(* Logix 5000 project; controller IF2_DEMO Emulate 5570 rev 20.12; software revision 20.04; part 2 of 8 *)
(* tags used below, declared in another part *)
   AlarmFillerConvJam : BOOL;
   ChangeOver_In_Progress : BOOL;
   Current_Order : STRING;
   CurrentCustomerName : STRING;
   CurrentPartName : STRING;
   DispenserLine : LineData;
   Filler_Stopped : BOOL;
   Labeler_Stopped : BOOL;
   Line1 : FTVPDemoLine;
   Next_Order : STRING;
   Next_Product : DINT;
   OEE_Part_Scrap_Old : DINT;
   OEE_Scrap_Filler : DINT;
   OrderQty : DINT[4];
   Packaging_Stopped : BOOL;
   PartCountRollOver : DINT;
   Previous_Order : STRING;
   PreviousCustomerName : STRING;
   PreviousPartName : STRING;
   ProdCounts : Counts;
   Product_Change : DINT;
   ProductionStart : BOOL;
   Starve_Block_Filler_Start_Toggle : BOOL;
   Starve_Block_Labeler_Start_Toggle : BOOL;
   Starve_Block_Packaging_Start_Toggle : BOOL;
   Timer1000ms : TIMER;
   Timer250ms : TIMER;
   WallClock : DINT[7];
   WC : WC[10];
   WorkOrder : WorkOrder;

PROGRAM FillerD   (* main routine MainRoutine *)
VAR
   Alarm_Filler1_Blocked : ALARM_DIGITAL;
   Alarm_Filler1_Starved : ALARM_DIGITAL;
   Alarm_Filler1_Stopped : ALARM_DIGITAL;
   ATest : BOOL;
   Block_Delay : TIMER := (PRE := 15000);
   Blocked_Condition : BOOL;
   Blocked_L : BOOL;
   BottleNum : STRING := '3';
   Change_Nextorder_name : BOOL;
   Change_order_name : BOOL;
   Ctrl_Bit : BOOL;
   DownStream_Run : ALIAS FOR WC[2].EventTrigger[0].1;
   DownStream_Running : ALIAS FOR WC[2].EventTrigger[0].8;
   Events : Events := (DownTime.Breakdown := 1, DownTime.BreakdownCode := 4, Control.StandbyCode := 1, Control.Auto := 1);
   Events_Control_Auto : ALIAS FOR WC_L.EventTrigger[0].5;
   Events_Control_OpStop : ALIAS FOR WC_L.EventTrigger[0].3;
   Events_Control_Run : ALIAS FOR WC_L.EventTrigger[0].1;
   Events_Control_Running : ALIAS FOR WC_L.EventTrigger[0].8;
   Events_Control_Standby : ALIAS FOR WC_L.EventTrigger[0].0;
   Events_Control_StandbyCode : ALIAS FOR WC_L.EventValue_REAL[1];
   Events_DownTime_Breakdown : ALIAS FOR WC_L.EventTrigger[0].2;
   Events_DownTime_BreakdownCode : ALIAS FOR WC_L.EventValue_REAL[2];
   Events_DownTime_Testing : ALIAS FOR WC_L.EventTrigger[0].7;
   Events_DownTime_UnschedMaint : ALIAS FOR WC_L.EventTrigger[0].6;
   Events_Operate_Load : ALIAS FOR WC_L.EventTrigger[0].10;
   Events_Operate_OrderProc : ALIAS FOR WC_L.EventTrigger[0].11;
   Events_Operate_Setup : ALIAS FOR WC_L.EventTrigger[0].9;
   Expected_Full_Production_Rate : DINT := 119;
   Filler : FTVPDemoWorkCell := (LineName := 'Line1', RunState := 1, Temperature := 95, ScrapRate := 6, ProductionRate := 119, Pressure := 123, OrderName := 'GF-08-CZ-525', CustomerName := 'Soda Inc.', PartName := 'GF-11');
   Filler_Start : BOOL := 1;
   Filler_State : DINT;
   Filler_Status : DINT := 1;
   Filler_Stop : BOOL;
   FillOunces : INT := 32;
   Force_Periodic_Changeover : DINT;
   HMI : HMIVars := (ScrapRate := 1.0, SpeedControl := 400.0, PrevSpeed := 100.0, CurrentProductionRate := 120.0, PartCountRollOver := 3500, MfgTimeBase := 1, MaxEventDur := 21.0, MinEventDur := 9.0, EventsPerHr := 100, EventDur := 20.688032, RunDur := 14.955534, MinRunDur := 5.0);
   MfgOrders : MfgOrders := (CustomerName := 'Big-Mart', OrderName := 'A123', ProdRate := 60.0, PartName := 'Apple-D12', WorkcellName := 'Filler 1', PartNameSav := 'Apple-D12');
   MfgOrders_CustomerName : ALIAS FOR WC_L.FlexSTRING[4];
   MfgOrders_Order : STRING := 'GF-08-CZ-525';
   MfgOrders_OrderName : ALIAS FOR WC_L.FlexSTRING[3];
   MfgOrders_OrderName_Blueberry : STRING := 'BL-03-RM-';
   MfgOrders_OrderName_Grapefruit : STRING := 'GF-08-CZ-';
   MfgOrders_OrderName_Kiwi : STRING := 'KW-05-JM-';
   MfgOrders_OrderName_Mango : STRING := 'MG-01-RZ-';
   MfgOrders_OrderNumber_Blueberry : DINT := 662;
   MfgOrders_OrderNumber_Grapefruit : DINT := 525;
   MfgOrders_OrderNumber_Kiwi : DINT := 651;
   MfgOrders_OrderNumber_Mango : DINT := 969;
   MfgOrders_OrderNumber_String : STRING := '970';
   MfgOrders_PartName : ALIAS FOR WC_L.FlexSTRING[0];
   Motion : DINT := 82;
   Motion_Counter : DINT := 1;
   Motion_Speed : DINT := 100;
   MotionCount : TIMER := (PRE := 9000, ACC := 8273, EN := 1, TT := 1);
   NA_Test : BOOL;
   New_Product_Change : BOOL;
   OEE : OEE := (IdealCycleTime := 5.0);
   OEE_IdealCycleTime : ALIAS FOR WC_L.IdealCT;
   OEE_Parts_Good : ALIAS FOR WC_L.GoodParts;
   OEE_Parts_Scrap : ALIAS FOR WC_L.ScrapParts;
   OEE_Parts_Total : ALIAS FOR WC_L.TotalParts;
   onsbits : DINT;
   OperatorID : ALIAS FOR WC_L.FlexREAL[1];
   Pressure1 : ALIAS FOR WC_L.PV[0];   // PSI
   ProductColor : DINT := 1;
   ProductColor_Save : DINT := 1;
   ProductColorCode : INT;
   RecipeFlag : BOOL;
   RecipeName : STRING := 'Super';
   SIM : SimVars := (Run.PRE := 14956, Event.PRE := 9000, Setup.PRE := 9000, Good := 2589.8208, Scrap := 26.160408, EventNumber := 11, UtilityBool[1] := 1, UtilityBool[2] := 1);
        .UTILITYBOOL[0]   // Enter Auto Mode ONS
        .UTILITYBOOL[1]   // Work Order Complete ONS
        .UTILITYBOOL[2]   // First Scan Bit
   skip : BOOL;
   Starve_Block_Filler_ONS : BOOL;
   Starve_Delay : TIMER := (PRE := 15000);
   Starved_L : BOOL;
   StateValue : ALIAS FOR WC_L.MonitorValue[0];
   Suppress : Events;
   Temperature1 : ALIAS FOR WC_L.PV[1];   // DEG
   TempReadTrigger : TIMER := (PRE := 5000, ACC := 3633, EN := 1, TT := 1);
   TempTimer : TIMER := (PRE := 10000, ACC := 3708, EN := 1, TT := 1);
   TempTimer2 : TIMER := (PRE := 5000, ACC := 3633, EN := 1, TT := 1);
   UpStream_Run : BOOL := 1;
   UpStream_Running : BOOL := 1;   // Not used-no upstream wc
   WC_L : ALIAS FOR WC[0];
END_VAR

ROUTINE MainRoutine   (* ladder *)
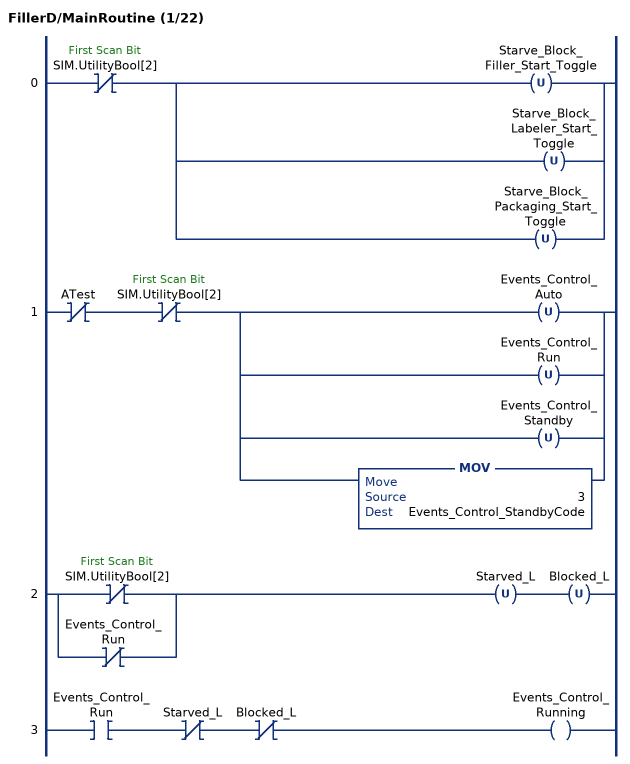
   0: XIO(SIM.UtilityBool[2])[OTU(Starve_Block_Filler_Start_Toggle) ,OTU(Starve_Block_Labeler_Start_Toggle) ,OTU(Starve_Block_Packaging_Start_Toggle) ];
   1: XIO(ATest)XIO(SIM.UtilityBool[2])[OTU(Events_Control_Auto) ,OTU(Events_Control_Run) ,OTU(Events_Control_Standby) ,MOV(3,Events_Control_StandbyCode) ];
   2: [XIO(SIM.UtilityBool[2]) ,XIO(Events_Control_Run) ]OTU(Starved_L)OTU(Blocked_L);
   3: XIC(Events_Control_Run)XIO(Starved_L)XIO(Blocked_L)OTE(Events_Control_Running);
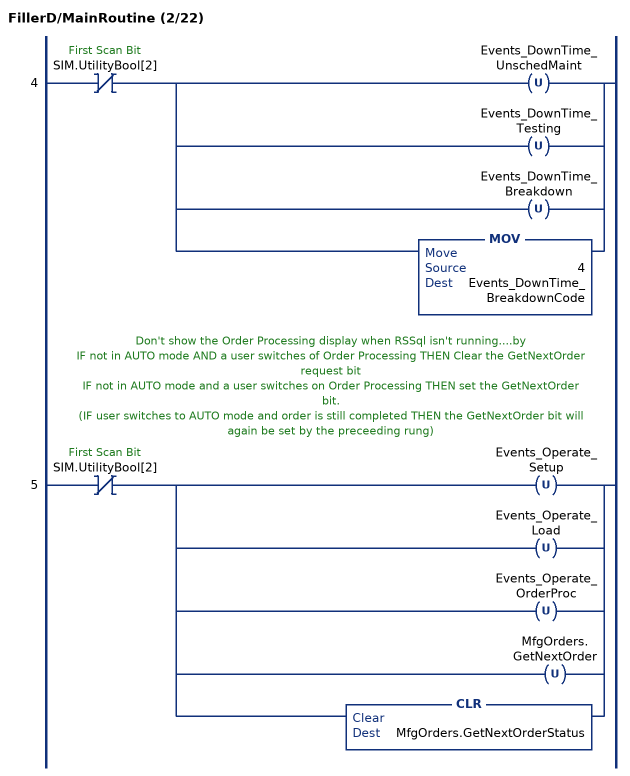
   4: XIO(SIM.UtilityBool[2])[OTU(Events_DownTime_UnschedMaint) ,OTU(Events_DownTime_Testing) ,OTU(Events_DownTime_Breakdown) ,MOV(4,Events_DownTime_BreakdownCode) ];
   // Don't show the Order Processing display when RSSql isn't running....by
   // IF not in AUTO mode AND a user switches of Order Processing THEN Clear the GetNextOrder request bit
   // IF not in AUTO mode and a user switches on Order Processing THEN set the GetNextOrder bit.
   // (IF user switches to AUTO mode and order is still completed THEN the GetNextOrder bit will again be set by the preceeding rung)
   5: XIO(SIM.UtilityBool[2])[OTU(Events_Operate_Setup) ,OTU(Events_Operate_Load) ,OTU(Events_Operate_OrderProc) ,OTU(MfgOrders.GetNextOrder) ,CLR(MfgOrders.GetNextOrderStatus) ];
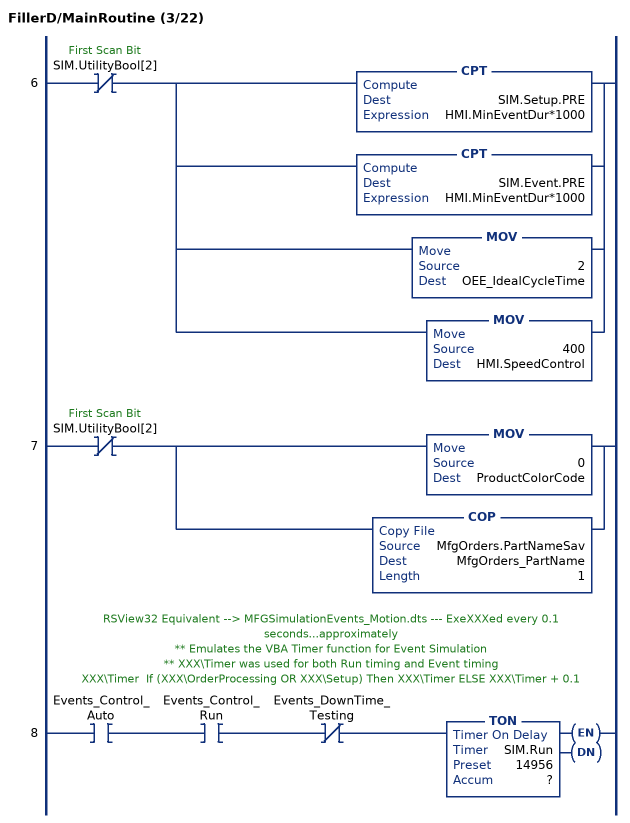
   6: XIO(SIM.UtilityBool[2])[CPT(SIM.Setup.PRE,HMI.MinEventDur*1000) ,CPT(SIM.Event.PRE,HMI.MinEventDur*1000) ,MOV(2,OEE_IdealCycleTime) ,MOV(400,HMI.SpeedControl) ];
   7: XIO(SIM.UtilityBool[2])[MOV(0,ProductColorCode) ,COP(MfgOrders.PartNameSav,MfgOrders_PartName,1) ];
   // RSView32 Equivalent --> MFGSimulationEvents_Motion.dts --- ExeXXXed every 0.1 seconds...approximately
   // ** Emulates the VBA Timer function for Event Simulation
   // ** XXX\Timer was used for both Run timing and Event timing
   // XXX\Timer	If (XXX\OrderProcessing OR XXX\Setup) Then XXX\Timer ELSE XXX\Timer + 0.1
   8: XIC(Events_Control_Auto)XIC(Events_Control_Run)XIO(Events_DownTime_Testing)TON(SIM.Run,?,?);
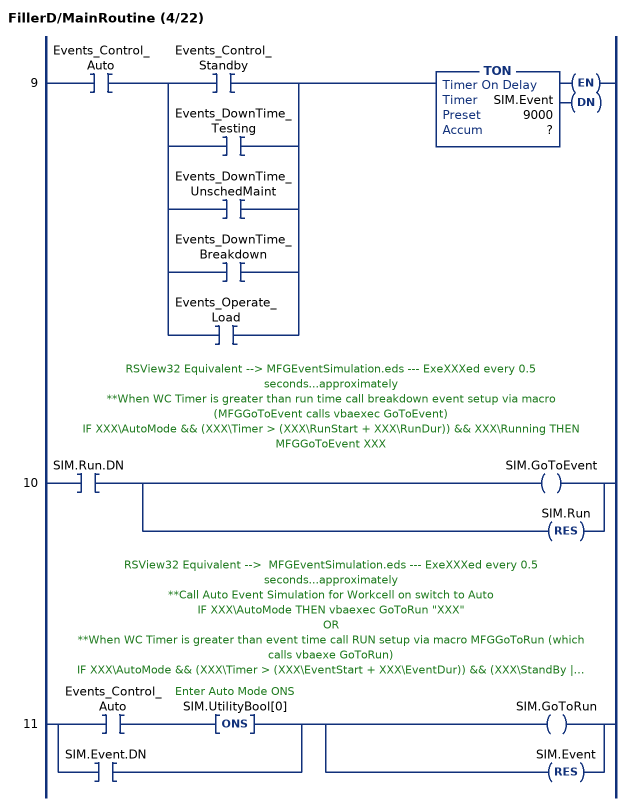
   9: XIC(Events_Control_Auto)[XIC(Events_Control_Standby) ,XIC(Events_DownTime_Testing) ,XIC(Events_DownTime_UnschedMaint) ,XIC(Events_DownTime_Breakdown) ,XIC(Events_Operate_Load) ]TON(SIM.Event,?,?);
   // RSView32 Equivalent --> MFGEventSimulation.eds --- ExeXXXed every 0.5 seconds...approximately
   // **When WC Timer is greater than run time call breakdown event setup via macro (MFGGoToEvent calls vbaexec GoToEvent)
   // IF XXX\AutoMode && (XXX\Timer > (XXX\RunStart + XXX\RunDur)) && XXX\Running THEN MFGGoToEvent XXX
   10: XIC(SIM.Run.DN)[OTE(SIM.GoToEvent) ,RES(SIM.Run) ];
   // RSView32 Equivalent -->  MFGEventSimulation.eds --- ExeXXXed every 0.5 seconds...approximately
   // **Call Auto Event Simulation for Workcell on switch to Auto
   // IF XXX\AutoMode THEN vbaexec GoToRun "XXX"
   // OR
   // **When WC Timer is greater than event time call RUN setup via macro MFGGoToRun (which calls vbaexe GoToRun)
   // IF XXX\AutoMode && (XXX\Timer > (XXX\EventStart + XXX\EventDur)) && (XXX\StandBy || XXX\Test || XXX\UnSchedMaint || XXX\Breakdown ||XXX\Load) THEN MFGGoToRun XXX
   11: [XIC(Events_Control_Auto) ONS(SIM.UtilityBool[0]) ,XIC(SIM.Event.DN) ][OTE(SIM.GoToRun) ,RES(SIM.Event) ];
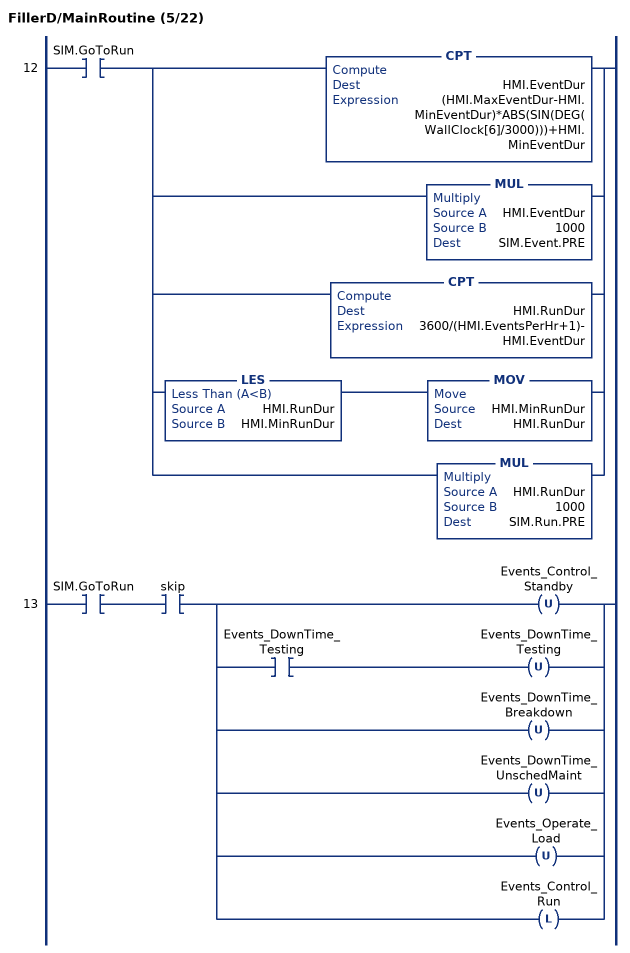
   12: XIC(SIM.GoToRun)[CPT(HMI.EventDur,(HMI.MaxEventDur-HMI.MinEventDur)*ABS(SIN(DEG(WallClock[6]/3000)))+HMI.MinEventDur) ,MUL(HMI.EventDur,1000,SIM.Event.PRE) ,CPT(HMI.RunDur,3600/(HMI.EventsPerHr+1)-HMI.EventDur) ,LES(HMI.RunDur,HMI.MinRunDur) MOV(HMI.MinRunDur,HMI.RunDur) ,MUL(HMI.RunDur,1000,SIM.Run.PRE) ];
   13: XIC(SIM.GoToRun)XIC(skip)[OTU(Events_Control_Standby) ,XIC(Events_DownTime_Testing) OTU(Events_DownTime_Testing) ,OTU(Events_DownTime_Breakdown) ,OTU(Events_DownTime_UnschedMaint) ,OTU(Events_Operate_Load) ,OTL(Events_Control_Run) ];
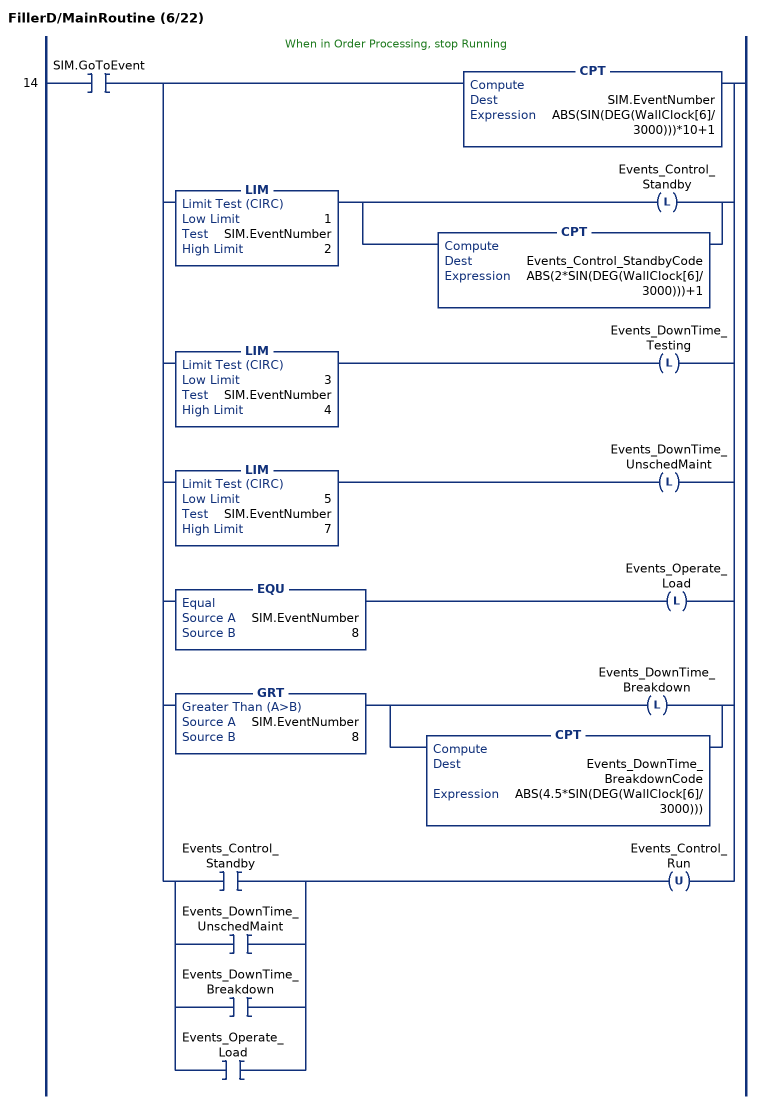
   // When in Order Processing, stop Running
   14: XIC(SIM.GoToEvent)[CPT(SIM.EventNumber,ABS(SIN(DEG(WallClock[6]/3000)))*10+1) ,LIM(1,SIM.EventNumber,2) [OTL(Events_Control_Standby) ,CPT(Events_Control_StandbyCode,ABS(2*SIN(DEG(WallClock[6]/3000)))+1) ] ,LIM(3,SIM.EventNumber,4) OTL(Events_DownTime_Testing) ,LIM(5,SIM.EventNumber,7) OTL(Events_DownTime_UnschedMaint) ,EQU(SIM.EventNumber,8) OTL(Events_Operate_Load) ,GRT(SIM.EventNumber,8) [OTL(Events_DownTime_Breakdown) ,CPT(Events_DownTime_BreakdownCode,ABS(4.5*SIN(DEG(WallClock[6]/3000)))) ] ,[XIC(Events_Control_Standby) ,XIC(Events_DownTime_UnschedMaint) ,XIC(Events_DownTime_Breakdown) ,XIC(Events_Operate_Load) ] OTU(Events_Control_Run) ];
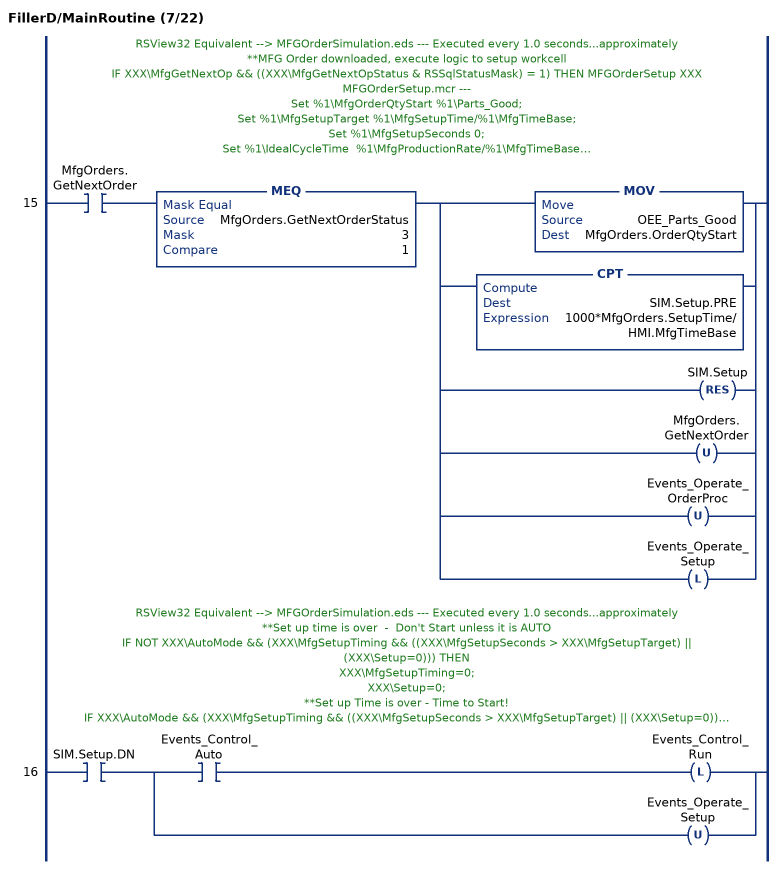
   // RSView32 Equivalent --> MFGOrderSimulation.eds --- Executed every 1.0 seconds...approximately
   // **MFG Order downloaded, execute logic to setup workcell
   // IF XXX\MfgGetNextOp && ((XXX\MfgGetNextOpStatus & RSSqlStatusMask) = 1) THEN MFGOrderSetup XXX
   // MFGOrderSetup.mcr ---
   // 	Set %1\MfgOrderQtyStart %1\Parts_Good;
   // 	Set %1\MfgSetupTarget %1\MfgSetupTime/%1\MfgTimeBase;
   // 	Set %1\MfgSetupSeconds 0;
   // 	Set %1\IdealCycleTime  %1\MfgProductionRate/%1\MfgTimeBase;
   // 	Set %1\MfgGetNextOp 0;
   // 	Set %1\Setup 1;
   // 	Set %1\OrderProcessing 0;
   // 	Set %1\MfgSetupTiming 1;
   15: XIC(MfgOrders.GetNextOrder)MEQ(MfgOrders.GetNextOrderStatus,3,1)[MOV(OEE_Parts_Good,MfgOrders.OrderQtyStart) ,CPT(SIM.Setup.PRE,1000*MfgOrders.SetupTime/HMI.MfgTimeBase) ,RES(SIM.Setup) ,OTU(MfgOrders.GetNextOrder) ,OTU(Events_Operate_OrderProc) ,OTL(Events_Operate_Setup) ];
   // RSView32 Equivalent --> MFGOrderSimulation.eds --- Executed every 1.0 seconds...approximately
   // **Set up time is over  -  Don't Start unless it is AUTO
   // IF NOT XXX\AutoMode && (XXX\MfgSetupTiming && ((XXX\MfgSetupSeconds > XXX\MfgSetupTarget) || (XXX\Setup=0))) THEN
   // 	XXX\MfgSetupTiming=0;
   // 	XXX\Setup=0;
   // **Set up Time is over - Time to Start!
   // IF XXX\AutoMode && (XXX\MfgSetupTiming && ((XXX\MfgSetupSeconds > XXX\MfgSetupTarget) || (XXX\Setup=0))) THEN
   // 	XXX\MfgSetupTiming=0;
   // 	XXX\Setup=0;
   // 	XXX\RUNNING=1
   16: XIC(SIM.Setup.DN)[XIC(Events_Control_Auto) OTL(Events_Control_Run) ,OTU(Events_Operate_Setup) ];
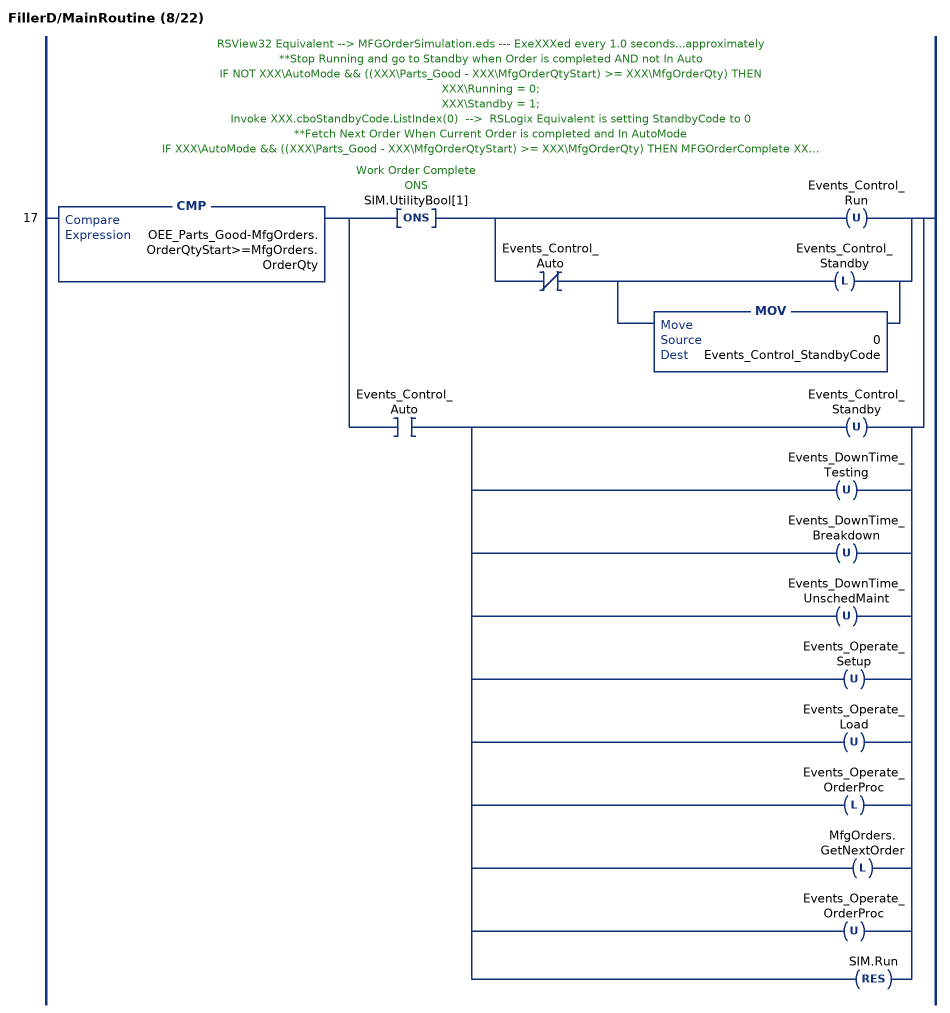
   // RSView32 Equivalent --> MFGOrderSimulation.eds --- ExeXXXed every 1.0 seconds...approximately
   // **Stop Running and go to Standby when Order is completed AND not In Auto
   // IF NOT XXX\AutoMode && ((XXX\Parts_Good - XXX\MfgOrderQtyStart) >= XXX\MfgOrderQty) THEN
   // 	XXX\Running = 0;
   // 	XXX\Standby = 1;
   // 	Invoke XXX.cboStandbyCode.ListIndex(0)  -->  RSLogix Equivalent is setting StandbyCode to 0
   // **Fetch Next Order When Current Order is completed and In AutoMode
   // IF XXX\AutoMode && ((XXX\Parts_Good - XXX\MfgOrderQtyStart) >= XXX\MfgOrderQty) THEN MFGOrderComplete XXX
   // MFGOrderComplete.mcr --- (Macros exeXXXed when called. %1 is the Workcell name -- typical all mcrs)
   // 	Set %1\RunStart %1\Timer;
   // 	Set %1\StandBy 0;
   // 	Set %1\Test 0;
   // 	Set %1\UnSchedMaint 0;
   // 	Set %1\Breakdown 0;
   // 	Set %1\Load 0;
   // 	Set %1\OrderProcessing 1;
   // 	Set %1\Running 0;
   // 	Set %1\MFGGetNextOpStatus 0;
   // 	Set %1\MFGGetNextOp 1
   17: CMP(OEE_Parts_Good-MfgOrders.OrderQtyStart>=MfgOrders.OrderQty)[ONS(SIM.UtilityBool[1]) [OTU(Events_Control_Run) ,XIO(Events_Control_Auto) [OTL(Events_Control_Standby) ,MOV(0,Events_Control_StandbyCode) ] ] ,XIC(Events_Control_Auto) [OTU(Events_Control_Standby) ,OTU(Events_DownTime_Testing) ,OTU(Events_DownTime_Breakdown) ,OTU(Events_DownTime_UnschedMaint) ,OTU(Events_Operate_Setup) ,OTU(Events_Operate_Load) ,OTL(Events_Operate_OrderProc) ,OTL(MfgOrders.GetNextOrder) ,OTU(Events_Operate_OrderProc) ,RES(SIM.Run) ] ];
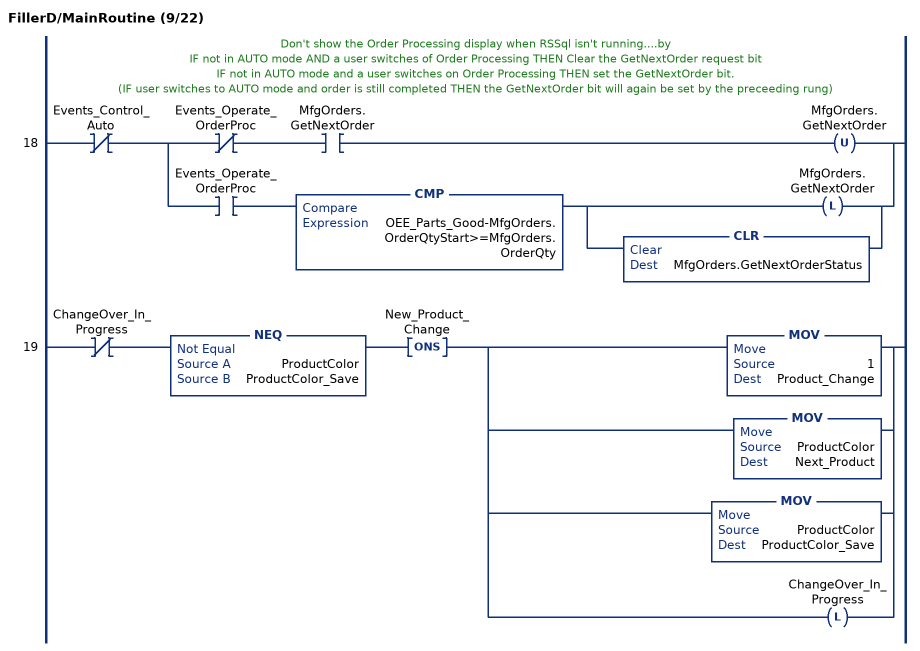
   // Don't show the Order Processing display when RSSql isn't running....by
   // IF not in AUTO mode AND a user switches of Order Processing THEN Clear the GetNextOrder request bit
   // IF not in AUTO mode and a user switches on Order Processing THEN set the GetNextOrder bit.
   // (IF user switches to AUTO mode and order is still completed THEN the GetNextOrder bit will again be set by the preceeding rung)
   18: XIO(Events_Control_Auto)[XIO(Events_Operate_OrderProc) XIC(MfgOrders.GetNextOrder) OTU(MfgOrders.GetNextOrder) ,XIC(Events_Operate_OrderProc) CMP(OEE_Parts_Good-MfgOrders.OrderQtyStart>=MfgOrders.OrderQty) [OTL(MfgOrders.GetNextOrder) ,CLR(MfgOrders.GetNextOrderStatus) ] ];
   19: XIO(ChangeOver_In_Progress)NEQ(ProductColor,ProductColor_Save)ONS(New_Product_Change)[MOV(1,Product_Change) ,MOV(ProductColor,Next_Product) ,MOV(ProductColor,ProductColor_Save) ,OTL(ChangeOver_In_Progress) ];
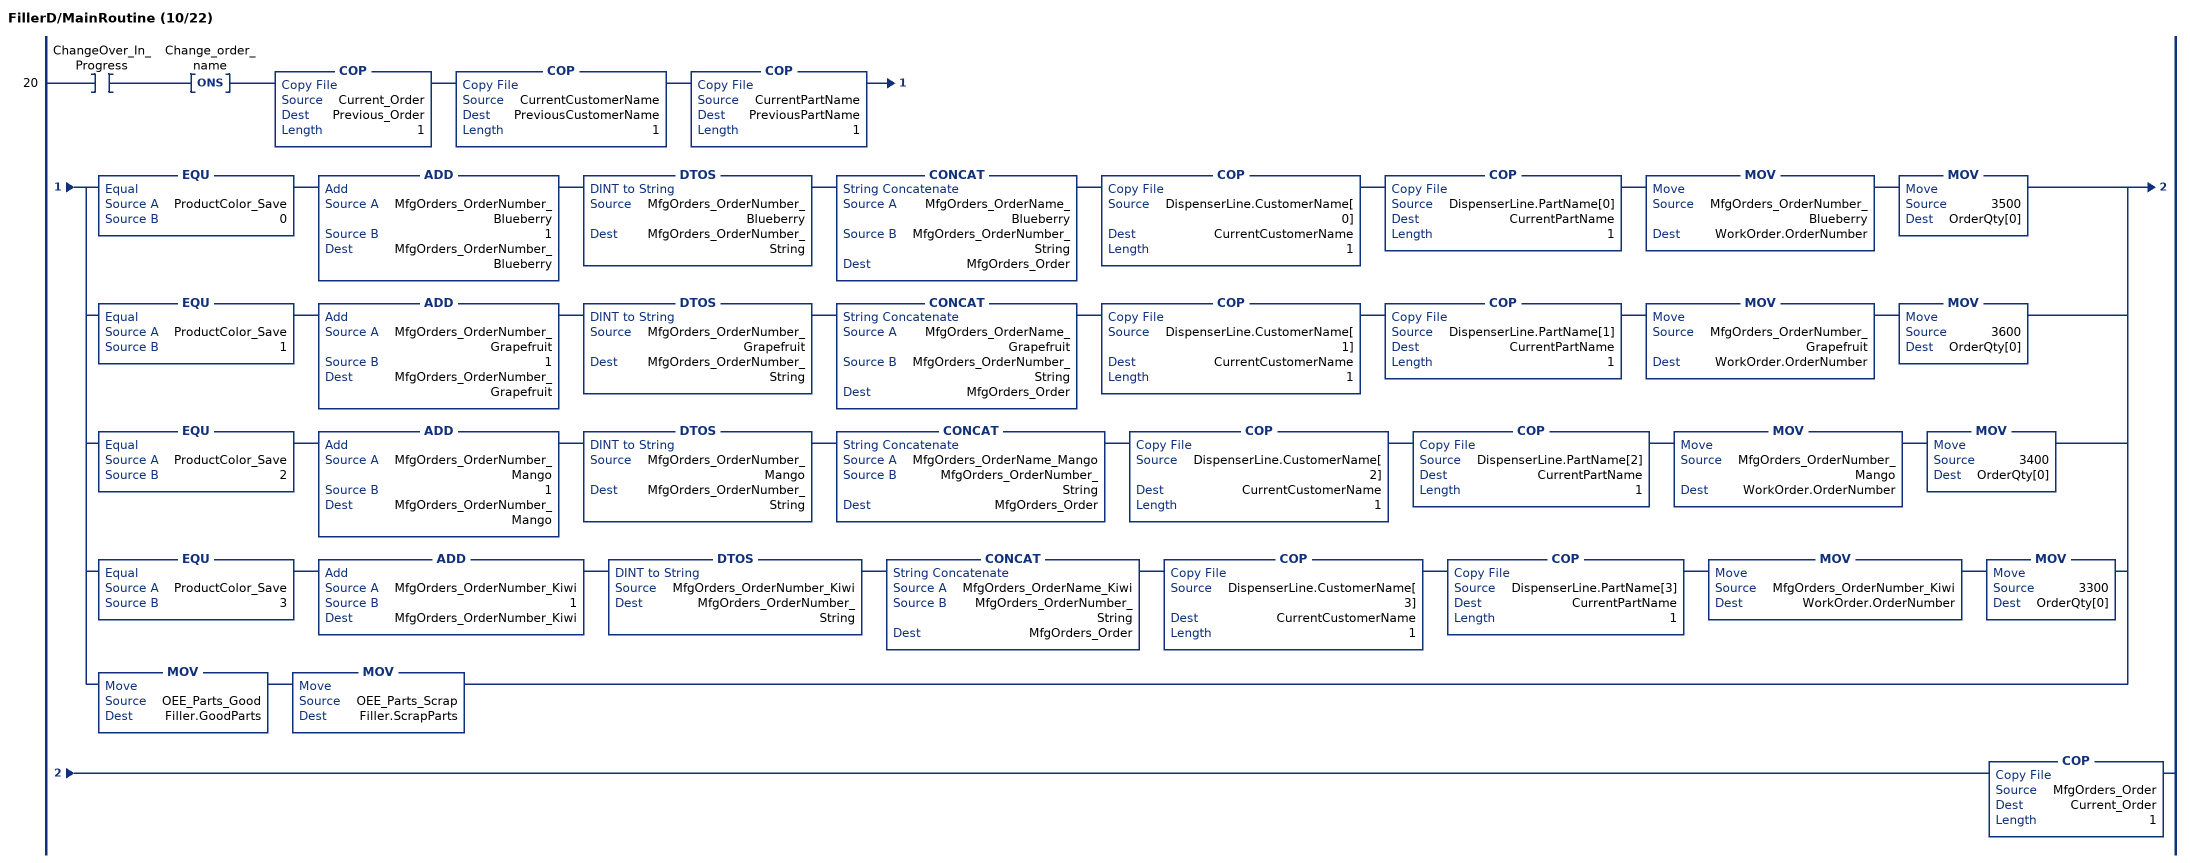
   20: XIC(ChangeOver_In_Progress)ONS(Change_order_name)COP(Current_Order,Previous_Order,1)COP(CurrentCustomerName,PreviousCustomerName,1)COP(CurrentPartName,PreviousPartName,1)[EQU(ProductColor_Save,0) ADD(MfgOrders_OrderNumber_Blueberry,1,MfgOrders_OrderNumber_Blueberry) DTOS(MfgOrders_OrderNumber_Blueberry,MfgOrders_OrderNumber_String) CONCAT(MfgOrders_OrderName_Blueberry,MfgOrders_OrderNumber_String,MfgOrders_Order) COP(DispenserLine.CustomerName[0],CurrentCustomerName,1) COP(DispenserLine.PartName[0],CurrentPartName,1) MOV(MfgOrders_OrderNumber_Blueberry,WorkOrder.OrderNumber) MOV(3500,OrderQty[0]) ,EQU(ProductColor_Save,1) ADD(MfgOrders_OrderNumber_Grapefruit,1,MfgOrders_OrderNumber_Grapefruit) DTOS(MfgOrders_OrderNumber_Grapefruit,MfgOrders_OrderNumber_String) CONCAT(MfgOrders_OrderName_Grapefruit,MfgOrders_OrderNumber_String,MfgOrders_Order) COP(DispenserLine.CustomerName[1],CurrentCustomerName,1) COP(DispenserLine.PartName[1],CurrentPartName,1) MOV(MfgOrders_OrderNumber_Grapefruit,WorkOrder.OrderNumber) MOV(3600,OrderQty[0]) ,EQU(ProductColor_Save,2) ADD(MfgOrders_OrderNumber_Mango,1,MfgOrders_OrderNumber_Mango) DTOS(MfgOrders_OrderNumber_Mango,MfgOrders_OrderNumber_String) CONCAT(MfgOrders_OrderName_Mango,MfgOrders_OrderNumber_String,MfgOrders_Order) COP(DispenserLine.CustomerName[2],CurrentCustomerName,1) COP(DispenserLine.PartName[2],CurrentPartName,1) MOV(MfgOrders_OrderNumber_Mango,WorkOrder.OrderNumber) MOV(3400,OrderQty[0]) ,EQU(ProductColor_Save,3) ADD(MfgOrders_OrderNumber_Kiwi,1,MfgOrders_OrderNumber_Kiwi) DTOS(MfgOrders_OrderNumber_Kiwi,MfgOrders_OrderNumber_String) CONCAT(MfgOrders_OrderName_Kiwi,MfgOrders_OrderNumber_String,MfgOrders_Order) COP(DispenserLine.CustomerName[3],CurrentCustomerName,1) COP(DispenserLine.PartName[3],CurrentPartName,1) MOV(MfgOrders_OrderNumber_Kiwi,WorkOrder.OrderNumber) MOV(3300,OrderQty[0]) ,MOV(OEE_Parts_Good,Filler.GoodParts) MOV(OEE_Parts_Scrap,Filler.ScrapParts) ]COP(MfgOrders_Order,Current_Order,1);
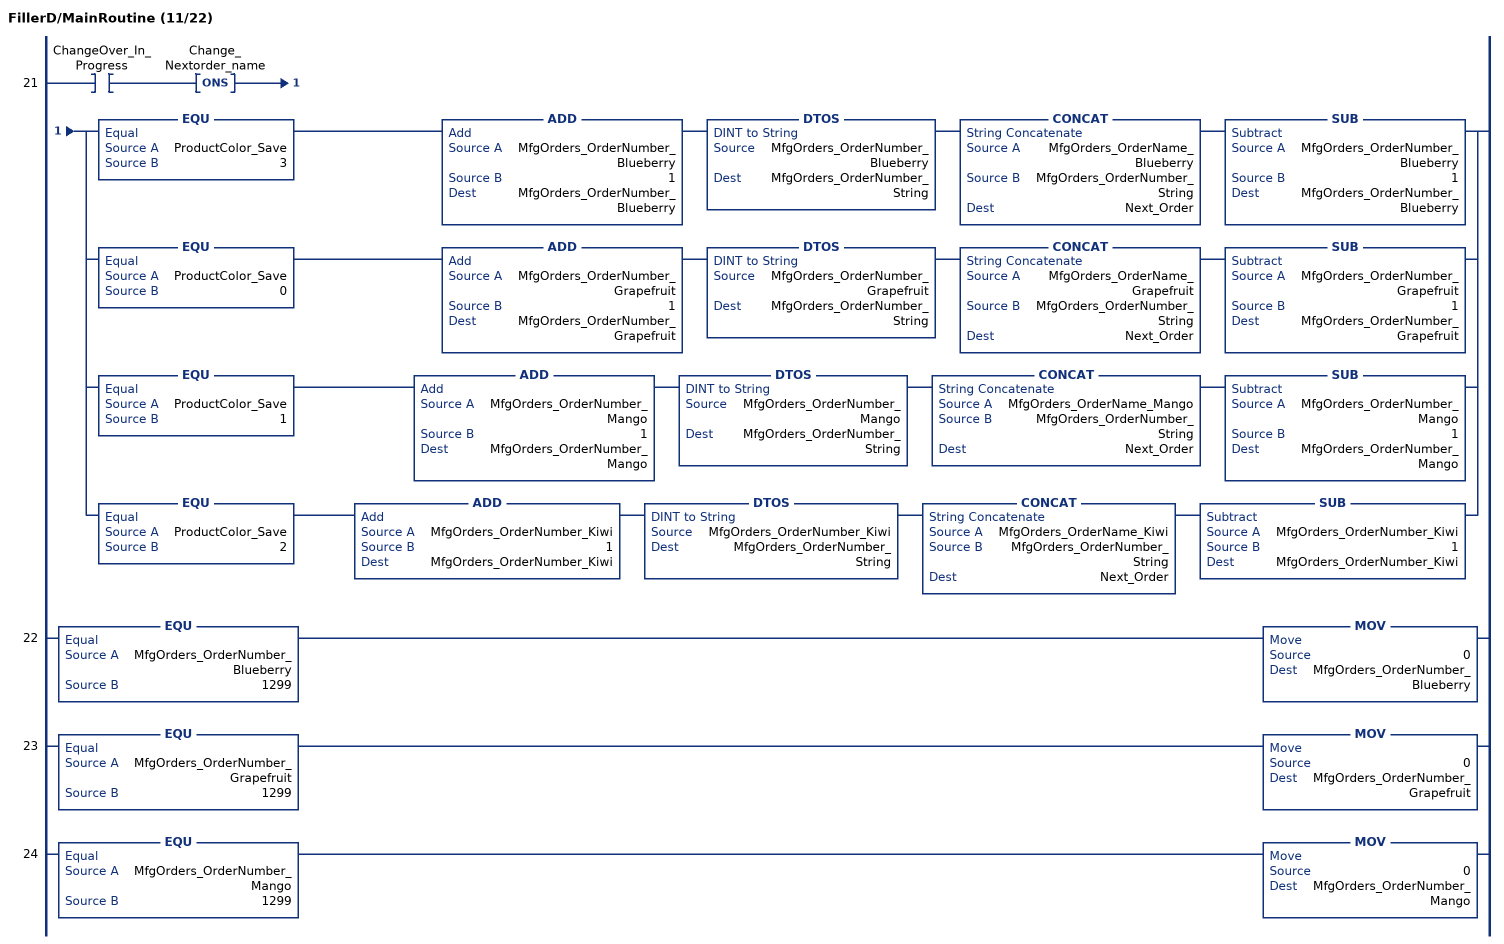
   21: XIC(ChangeOver_In_Progress)ONS(Change_Nextorder_name)[EQU(ProductColor_Save,3) ADD(MfgOrders_OrderNumber_Blueberry,1,MfgOrders_OrderNumber_Blueberry) DTOS(MfgOrders_OrderNumber_Blueberry,MfgOrders_OrderNumber_String) CONCAT(MfgOrders_OrderName_Blueberry,MfgOrders_OrderNumber_String,Next_Order) SUB(MfgOrders_OrderNumber_Blueberry,1,MfgOrders_OrderNumber_Blueberry) ,EQU(ProductColor_Save,0) ADD(MfgOrders_OrderNumber_Grapefruit,1,MfgOrders_OrderNumber_Grapefruit) DTOS(MfgOrders_OrderNumber_Grapefruit,MfgOrders_OrderNumber_String) CONCAT(MfgOrders_OrderName_Grapefruit,MfgOrders_OrderNumber_String,Next_Order) SUB(MfgOrders_OrderNumber_Grapefruit,1,MfgOrders_OrderNumber_Grapefruit) ,EQU(ProductColor_Save,1) ADD(MfgOrders_OrderNumber_Mango,1,MfgOrders_OrderNumber_Mango) DTOS(MfgOrders_OrderNumber_Mango,MfgOrders_OrderNumber_String) CONCAT(MfgOrders_OrderName_Mango,MfgOrders_OrderNumber_String,Next_Order) SUB(MfgOrders_OrderNumber_Mango,1,MfgOrders_OrderNumber_Mango) ,EQU(ProductColor_Save,2) ADD(MfgOrders_OrderNumber_Kiwi,1,MfgOrders_OrderNumber_Kiwi) DTOS(MfgOrders_OrderNumber_Kiwi,MfgOrders_OrderNumber_String) CONCAT(MfgOrders_OrderName_Kiwi,MfgOrders_OrderNumber_String,Next_Order) SUB(MfgOrders_OrderNumber_Kiwi,1,MfgOrders_OrderNumber_Kiwi) ];
   22: EQU(MfgOrders_OrderNumber_Blueberry,1299)MOV(0,MfgOrders_OrderNumber_Blueberry);
   23: EQU(MfgOrders_OrderNumber_Grapefruit,1299)MOV(0,MfgOrders_OrderNumber_Grapefruit);
   24: EQU(MfgOrders_OrderNumber_Mango,1299)MOV(0,MfgOrders_OrderNumber_Mango);
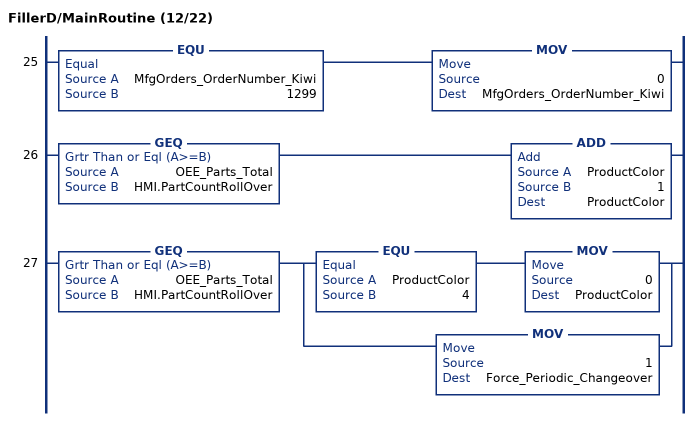
   25: EQU(MfgOrders_OrderNumber_Kiwi,1299)MOV(0,MfgOrders_OrderNumber_Kiwi);
   26: GEQ(OEE_Parts_Total,HMI.PartCountRollOver)ADD(ProductColor,1,ProductColor);
   27: GEQ(OEE_Parts_Total,HMI.PartCountRollOver)[EQU(ProductColor,4) MOV(0,ProductColor) ,MOV(1,Force_Periodic_Changeover) ];
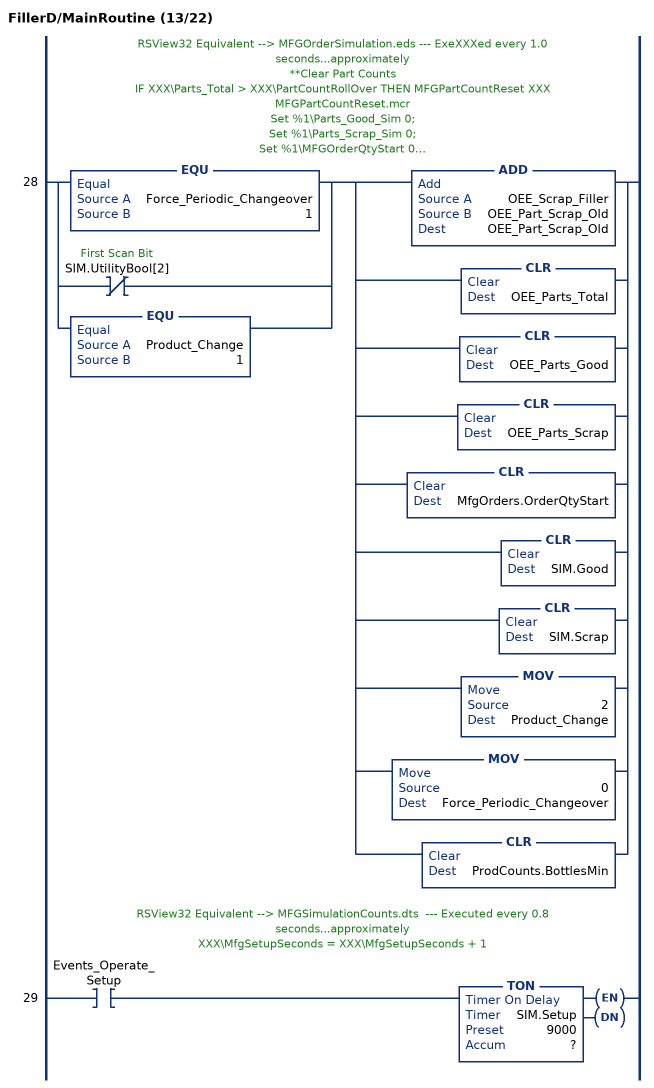
   // RSView32 Equivalent --> MFGOrderSimulation.eds --- ExeXXXed every 1.0 seconds...approximately
   // **Clear Part Counts
   // IF XXX\Parts_Total > XXX\PartCountRollOver THEN MFGPartCountReset XXX
   // MFGPartCountReset.mcr
   // 	Set %1\Parts_Good_Sim 0;
   // 	Set %1\Parts_Scrap_Sim 0;
   // 	Set %1\MFGOrderQtyStart 0;
   // 	Set %1\Parts_Good 0;
   // 	Set %1\Parts_Scrap 0;
   // 	Set %1\Parts_Total 0
   28: [EQU(Force_Periodic_Changeover,1) ,XIO(SIM.UtilityBool[2]) ,EQU(Product_Change,1) ][ADD(OEE_Scrap_Filler,OEE_Part_Scrap_Old,OEE_Part_Scrap_Old) ,CLR(OEE_Parts_Total) ,CLR(OEE_Parts_Good) ,CLR(OEE_Parts_Scrap) ,CLR(MfgOrders.OrderQtyStart) ,CLR(SIM.Good) ,CLR(SIM.Scrap) ,MOV(2,Product_Change) ,MOV(0,Force_Periodic_Changeover) ,CLR(ProdCounts.BottlesMin) ];
   // RSView32 Equivalent --> MFGSimulationCounts.dts	--- Executed every 0.8 seconds...approximately
   // XXX\MfgSetupSeconds = XXX\MfgSetupSeconds + 1
   29: XIC(Events_Operate_Setup)TON(SIM.Setup,?,?);
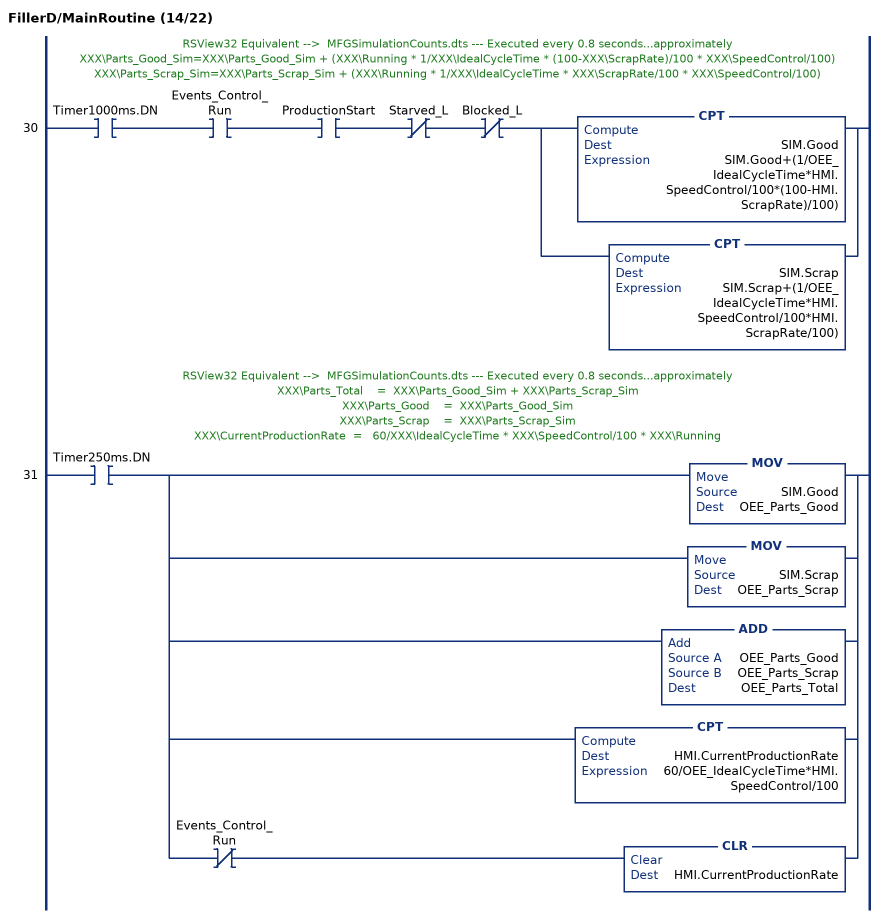
   // RSView32 Equivalent -->  MFGSimulationCounts.dts --- Executed every 0.8 seconds...approximately
   // XXX\Parts_Good_Sim=XXX\Parts_Good_Sim + (XXX\Running * 1/XXX\IdealCycleTime * (100-XXX\ScrapRate)/100 * XXX\SpeedControl/100)
   // XXX\Parts_Scrap_Sim=XXX\Parts_Scrap_Sim + (XXX\Running * 1/XXX\IdealCycleTime * XXX\ScrapRate/100 * XXX\SpeedControl/100)
   30: XIC(Timer1000ms.DN)XIC(Events_Control_Run)XIC(ProductionStart)XIO(Starved_L)XIO(Blocked_L)[CPT(SIM.Good,SIM.Good+(1/OEE_IdealCycleTime*HMI.SpeedControl/100*(100-HMI.ScrapRate)/100)) ,CPT(SIM.Scrap,SIM.Scrap+(1/OEE_IdealCycleTime*HMI.SpeedControl/100*HMI.ScrapRate/100)) ];
   // RSView32 Equivalent -->  MFGSimulationCounts.dts --- Executed every 0.8 seconds...approximately
   // XXX\Parts_Total		=	XXX\Parts_Good_Sim + XXX\Parts_Scrap_Sim
   // XXX\Parts_Good		=	XXX\Parts_Good_Sim
   // XXX\Parts_Scrap		=	XXX\Parts_Scrap_Sim
   // XXX\CurrentProductionRate  = 	60/XXX\IdealCycleTime * XXX\SpeedControl/100 * XXX\Running
   31: XIC(Timer250ms.DN)[[MOV(SIM.Good,OEE_Parts_Good) ,MOV(SIM.Scrap,OEE_Parts_Scrap) ,ADD(OEE_Parts_Good,OEE_Parts_Scrap,OEE_Parts_Total) ] ,CPT(HMI.CurrentProductionRate,60/OEE_IdealCycleTime*HMI.SpeedControl/100) ,XIO(Events_Control_Run) CLR(HMI.CurrentProductionRate) ];
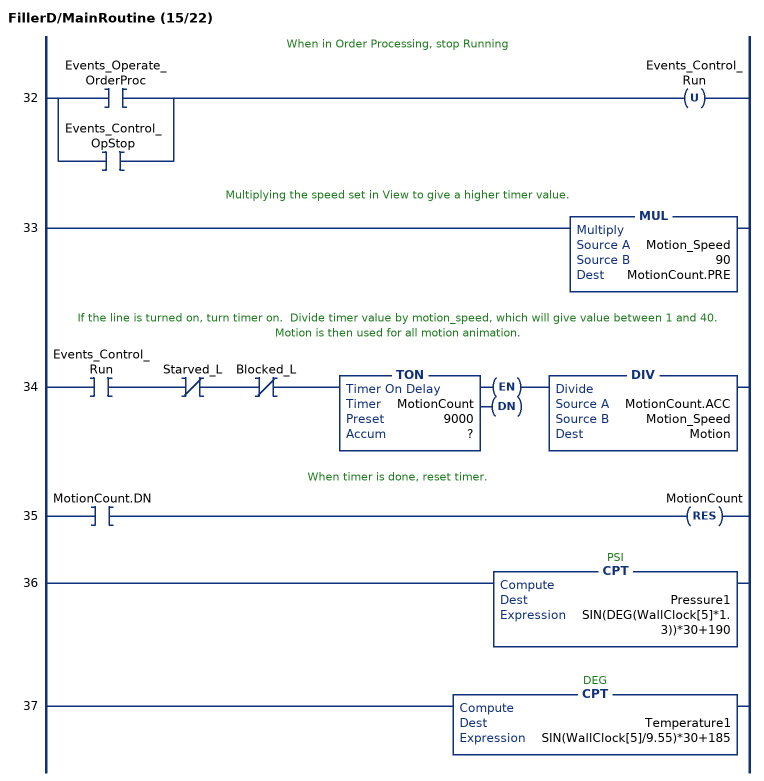
   // When in Order Processing, stop Running
   32: [XIC(Events_Operate_OrderProc) ,XIC(Events_Control_OpStop) ]OTU(Events_Control_Run);
   // Multiplying the speed set in View to give a higher timer value.
   33: MUL(Motion_Speed,90,MotionCount.PRE);
   // If the line is turned on, turn timer on.  Divide timer value by motion_speed, which will give value between 1 and 40.  Motion is then used for all motion animation.
   34: XIC(Events_Control_Run)XIO(Starved_L)XIO(Blocked_L)TON(MotionCount,?,?)DIV(MotionCount.ACC,Motion_Speed,Motion);
   // When timer is done, reset timer.
   35: XIC(MotionCount.DN)RES(MotionCount);
   36: CPT(Pressure1,SIN(DEG(WallClock[5]*1.3))*30+190);
   37: CPT(Temperature1,SIN(WallClock[5]/9.55)*30+185);
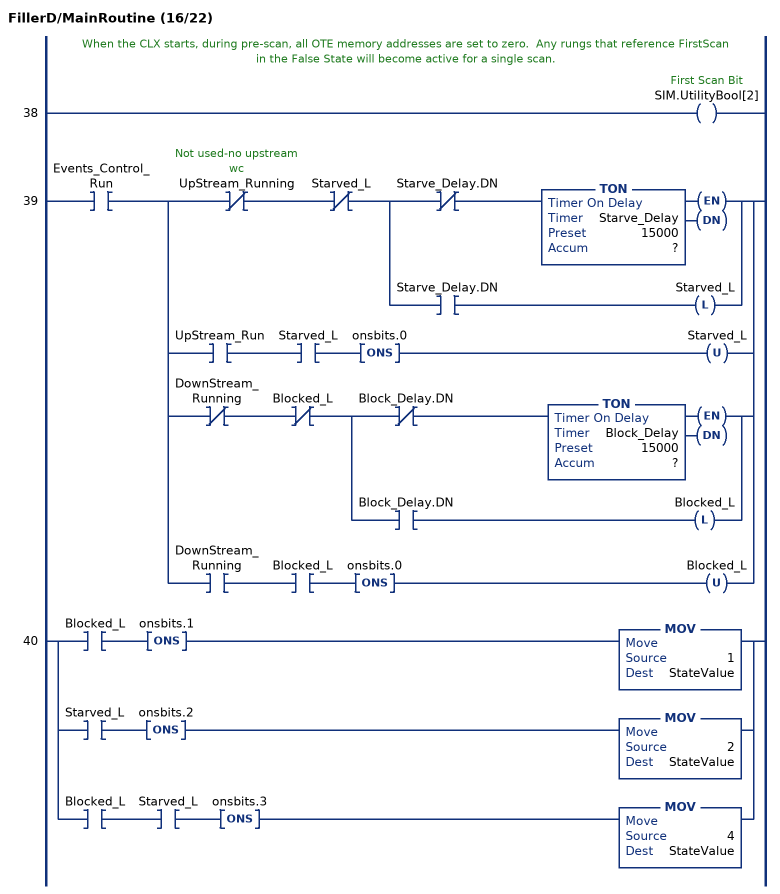
   // When the CLX starts, during pre-scan, all OTE memory addresses are set to zero.  Any rungs that reference FirstScan in the False State will become active for a single scan.
   38: OTE(SIM.UtilityBool[2]);
   39: XIC(Events_Control_Run)[[XIO(UpStream_Running) XIO(Starved_L) [XIO(Starve_Delay.DN) TON(Starve_Delay,?,?) ,XIC(Starve_Delay.DN) OTL(Starved_L) ] ,XIC(UpStream_Run) XIC(Starved_L) ONS(onsbits.0) OTU(Starved_L) ] ,[XIO(DownStream_Running) XIO(Blocked_L) [XIO(Block_Delay.DN) TON(Block_Delay,?,?) ,XIC(Block_Delay.DN) OTL(Blocked_L) ] ,XIC(DownStream_Running) XIC(Blocked_L) ONS(onsbits.0) OTU(Blocked_L) ] ];
   40: [XIC(Blocked_L) ONS(onsbits.1) MOV(1,StateValue) ,XIC(Starved_L) ONS(onsbits.2) MOV(2,StateValue) ,XIC(Blocked_L) XIC(Starved_L) ONS(onsbits.3) MOV(4,StateValue) ];
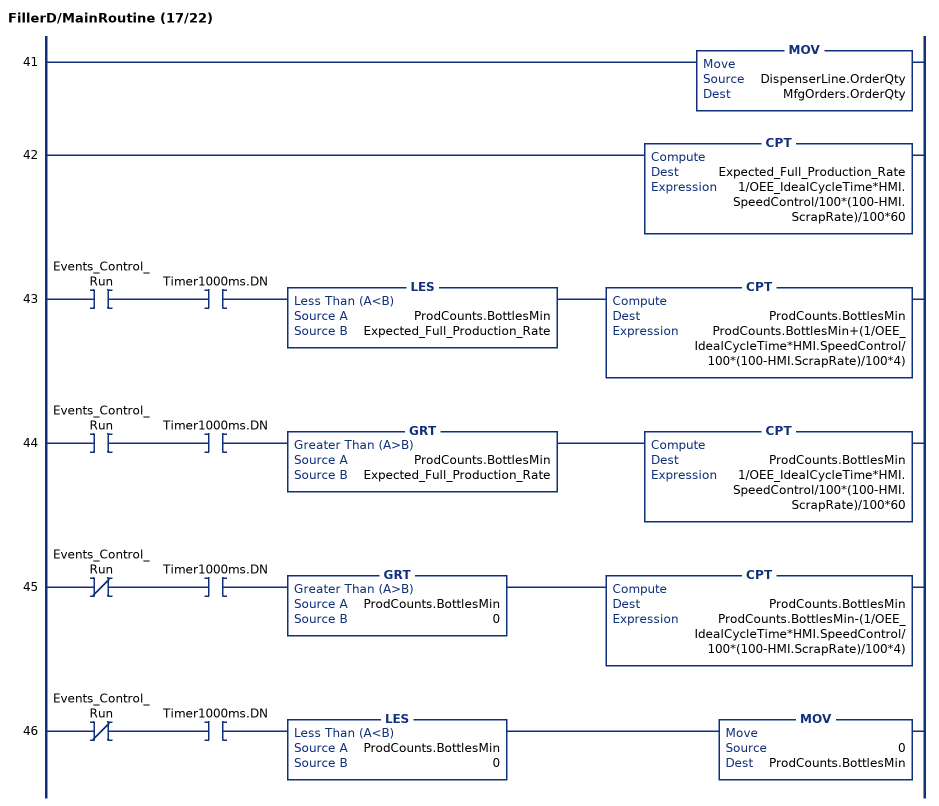
   41: MOV(DispenserLine.OrderQty,MfgOrders.OrderQty);
   42: CPT(Expected_Full_Production_Rate,1/OEE_IdealCycleTime*HMI.SpeedControl/100*(100-HMI.ScrapRate)/100*60);
   43: XIC(Events_Control_Run)XIC(Timer1000ms.DN)LES(ProdCounts.BottlesMin,Expected_Full_Production_Rate)CPT(ProdCounts.BottlesMin,ProdCounts.BottlesMin+(1/OEE_IdealCycleTime*HMI.SpeedControl/100*(100-HMI.ScrapRate)/100*4));
   44: XIC(Events_Control_Run)XIC(Timer1000ms.DN)GRT(ProdCounts.BottlesMin,Expected_Full_Production_Rate)CPT(ProdCounts.BottlesMin,1/OEE_IdealCycleTime*HMI.SpeedControl/100*(100-HMI.ScrapRate)/100*60);
   45: XIO(Events_Control_Run)XIC(Timer1000ms.DN)GRT(ProdCounts.BottlesMin,0)CPT(ProdCounts.BottlesMin,ProdCounts.BottlesMin-(1/OEE_IdealCycleTime*HMI.SpeedControl/100*(100-HMI.ScrapRate)/100*4));
   46: XIO(Events_Control_Run)XIC(Timer1000ms.DN)LES(ProdCounts.BottlesMin,0)MOV(0,ProdCounts.BottlesMin);
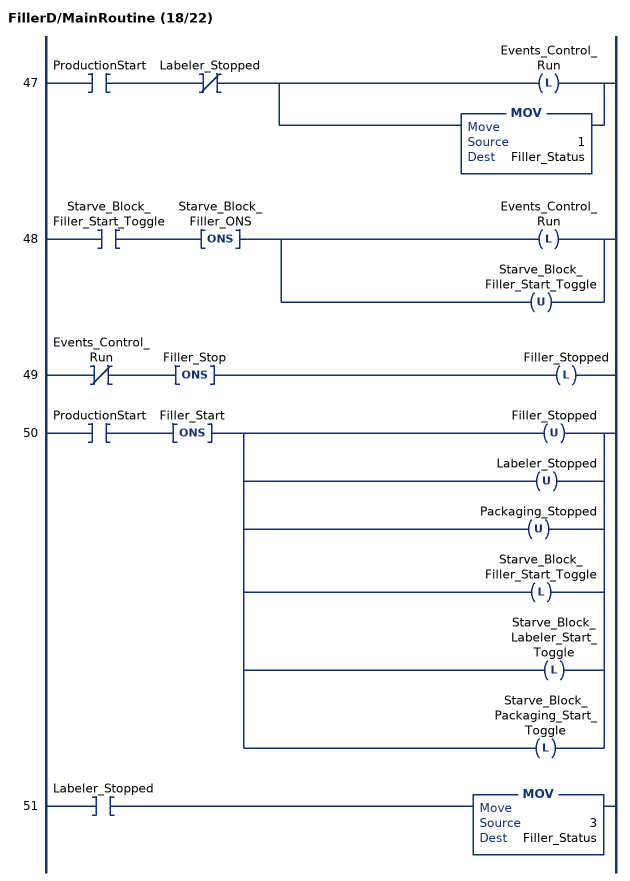
   47: XIC(ProductionStart)XIO(Labeler_Stopped)[OTL(Events_Control_Run) ,MOV(1,Filler_Status) ];
   48: XIC(Starve_Block_Filler_Start_Toggle)ONS(Starve_Block_Filler_ONS)[OTL(Events_Control_Run) ,OTU(Starve_Block_Filler_Start_Toggle) ];
   49: XIO(Events_Control_Run)ONS(Filler_Stop)OTL(Filler_Stopped);
   50: XIC(ProductionStart)ONS(Filler_Start)[OTU(Filler_Stopped) ,OTU(Labeler_Stopped) ,OTU(Packaging_Stopped) ,OTL(Starve_Block_Filler_Start_Toggle) ,OTL(Starve_Block_Labeler_Start_Toggle) ,OTL(Starve_Block_Packaging_Start_Toggle) ];
   51: XIC(Labeler_Stopped)MOV(3,Filler_Status);
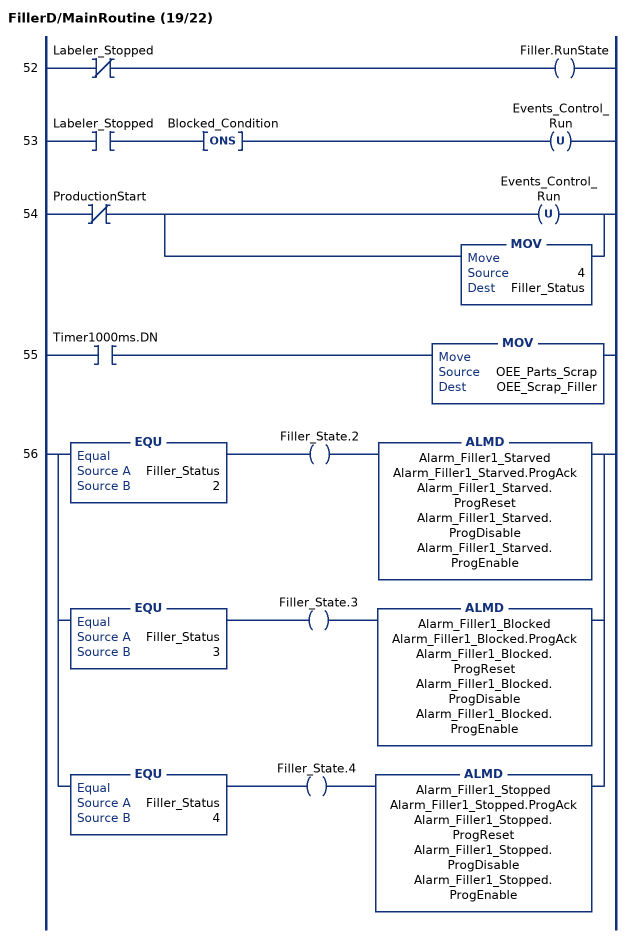
   52: XIO(Labeler_Stopped)OTE(Filler.RunState);
   53: XIC(Labeler_Stopped)ONS(Blocked_Condition)OTU(Events_Control_Run);
   54: XIO(ProductionStart)[OTU(Events_Control_Run) ,MOV(4,Filler_Status) ];
   55: XIC(Timer1000ms.DN)MOV(OEE_Parts_Scrap,OEE_Scrap_Filler);
   56: [EQU(Filler_Status,2) OTE(Filler_State.2) ALMD(Alarm_Filler1_Starved,Alarm_Filler1_Starved.ProgAck,Alarm_Filler1_Starved.ProgReset,Alarm_Filler1_Starved.ProgDisable,Alarm_Filler1_Starved.ProgEnable) ,EQU(Filler_Status,3) OTE(Filler_State.3) ALMD(Alarm_Filler1_Blocked,Alarm_Filler1_Blocked.ProgAck,Alarm_Filler1_Blocked.ProgReset,Alarm_Filler1_Blocked.ProgDisable,Alarm_Filler1_Blocked.ProgEnable) ,EQU(Filler_Status,4) OTE(Filler_State.4) ALMD(Alarm_Filler1_Stopped,Alarm_Filler1_Stopped.ProgAck,Alarm_Filler1_Stopped.ProgReset,Alarm_Filler1_Stopped.ProgDisable,Alarm_Filler1_Stopped.ProgEnable) ];
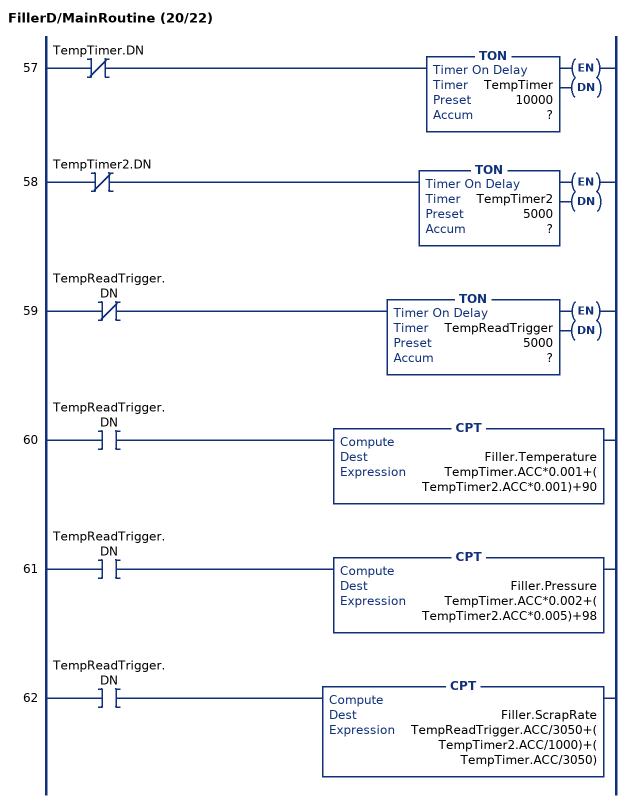
   57: XIO(TempTimer.DN)TON(TempTimer,?,?);
   58: XIO(TempTimer2.DN)TON(TempTimer2,?,?);
   59: XIO(TempReadTrigger.DN)TON(TempReadTrigger,?,?);
   60: XIC(TempReadTrigger.DN)CPT(Filler.Temperature,TempTimer.ACC*0.001+(TempTimer2.ACC*0.001)+90);
   61: XIC(TempReadTrigger.DN)CPT(Filler.Pressure,TempTimer.ACC*0.002+(TempTimer2.ACC*0.005)+98);
   62: XIC(TempReadTrigger.DN)CPT(Filler.ScrapRate,TempReadTrigger.ACC/3050+(TempTimer2.ACC/1000)+(TempTimer.ACC/3050));
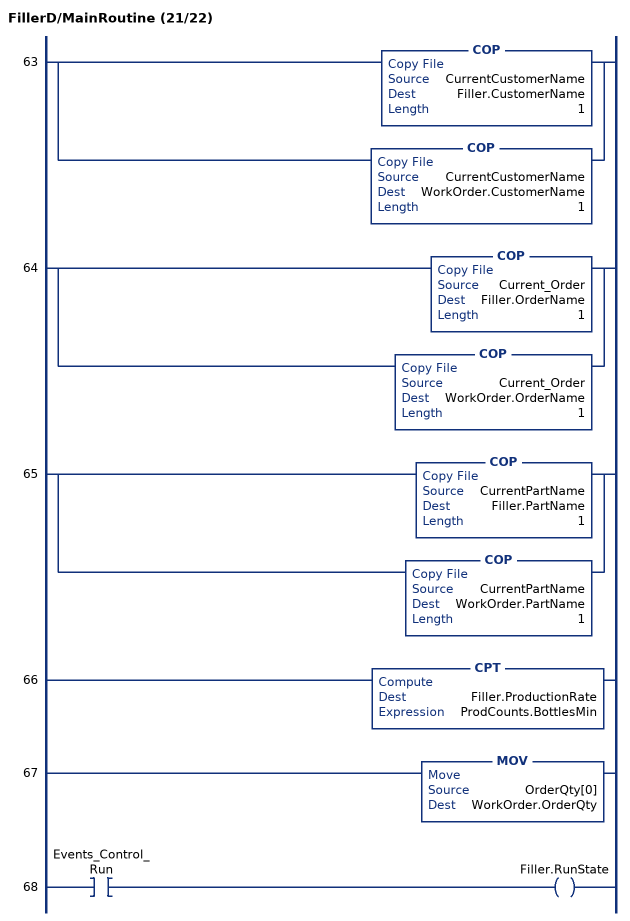
   63: [COP(CurrentCustomerName,Filler.CustomerName,1) ,COP(CurrentCustomerName,WorkOrder.CustomerName,1) ];
   64: [COP(Current_Order,Filler.OrderName,1) ,COP(Current_Order,WorkOrder.OrderName,1) ];
   65: [COP(CurrentPartName,Filler.PartName,1) ,COP(CurrentPartName,WorkOrder.PartName,1) ];
   66: CPT(Filler.ProductionRate,ProdCounts.BottlesMin);
   67: MOV(OrderQty[0],WorkOrder.OrderQty);
   68: XIC(Events_Control_Run)OTE(Filler.RunState);
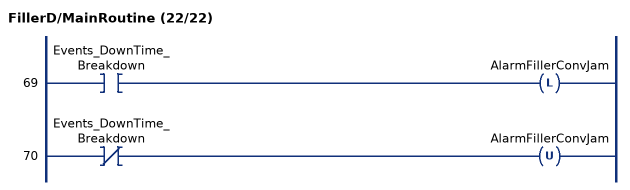
   69: XIC(Events_DownTime_Breakdown)OTL(AlarmFillerConvJam);
   70: XIO(Events_DownTime_Breakdown)OTU(AlarmFillerConvJam);
END_ROUTINE
END_PROGRAM
